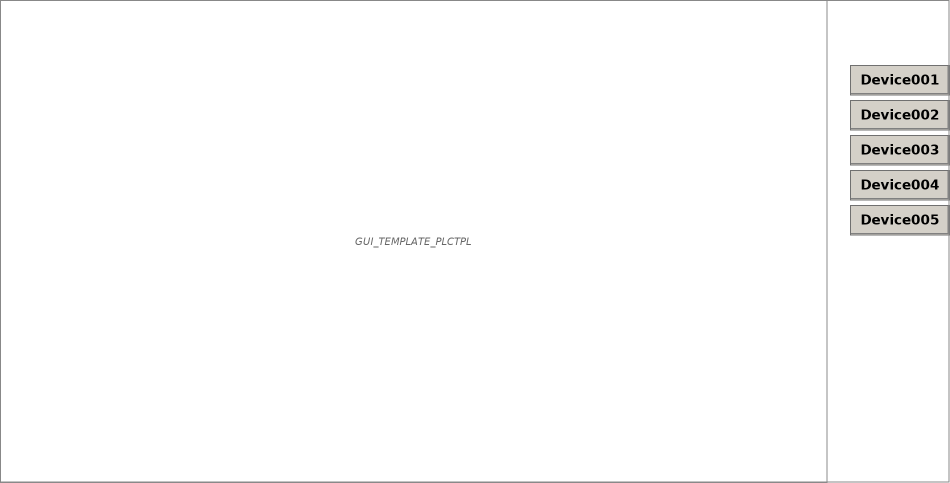
VISUALIZATION GUI_All  // 950x483
    Frame (0,0 827x483)
        shows GUI_TEMPLATE_PLCTPL(m_Instance := MAIN.ptrGUI_Devices[MAIN.nPtrIndex_Devices]^)
    Button (850,65 100x30), "Device001"
        OnMouseClick: execute { MAIN.nPtrIndex_Devices:=1; }
    Button (850,100 100x30), "Device002"
        OnMouseClick: execute { MAIN.nPtrIndex_Devices:=2; }
    Button (850,135 100x30), "Device003"
        OnMouseClick: execute { MAIN.nPtrIndex_Devices:=3; }
    Button (850,170 100x30), "Device004"
        OnMouseClick: execute { MAIN.nPtrIndex_Devices:=4; }
    Button (850,205 100x30), "Device005"
        OnMouseClick: execute { MAIN.nPtrIndex_Devices:=5; }
END_VISUALIZATION

(* stored: Version 1.1.0.1, ProductVersion 3.1.4024.3
   Visu GUI_All: Id {ba6b4829-cfe8-4c1b-80a7-d8c3b6d4dc60} *)
